(* Logix 5000 project; controller cal1615 1756-L62 rev 20.19; software revision 20.05; part 21 of 82 *)
(* tags used below, declared in another part *)
   AFI : BOOL;   // Always False Bit
   FAULT : BOOL;   // Fault AFI
   p01_param_fan_zero_speed : REAL;
   p01_param_open_oven_exh_sp : REAL;
   p01_recipe_active : recipe;   // Active Recipe
   p01r02 : routine;   // System Misc Control
   p01r09_open_oven : BOOL;
   p01r09_pb_global_reset : BOOL;   // System Modes PB: Global Fault Reset
   p02_dint_from_hmi : hmi_dint;
   p11_ai_exh_rpm : REAL;   // Zone 1 Analog Input Exhaust Fan RPM
   p11_ai_lfl : REAL;   // Zone 1 Analog Input Lower Flash Limit
   p11_ao_cv : REAL;   // Zone 1 Analog Output Control Valve
   p11_ao_exhaust_selected_speed : REAL;   // Zone 1 Analog Output Exhaust Fan VFD Selected Speed
   p11_di_burner_auto : BOOL;   // Zone 1 Digital Input Burner Auto
   p11_di_burner_safeties_ok : BOOL;   // Zone 1 Digital Input Burner Safeties Ok
   p11_di_door_open : BOOL;   // Zone 1 Digital Input Access Door Open
   p11_di_exh : acs800_di_normal;   // Zone 1 Digital Inputs Exhaust Fan
   p11_di_exh_fan_mtr_ts : BOOL;   // Zone 1 Digital Input Exhaust Fan Motor Thermostat OK
   p11_di_exh_flow_ok : BOOL;   // Zone 1 Digital Input Exhaust Flow OK
   p11_di_flame_failure : BOOL;   // Zone 1 Digital Input Flame Failure
   p11_di_flame_on : BOOL;   // Zone 1 Digital Input Burner is On
   p11_di_fresh_air_clean : BOOL;   // Zone 1 Digital Input Fresh Air Filter Dirty
   p11_di_high_limit_temp_ok : BOOL;   // Zone 1 Digital Input High Limit Temperature OK
   p11_di_recirc : acs800_di_normal;   // Zone 1 Digital Inputs Recirc Fan
   p11_di_recirc_flow_ok : BOOL;   // Zone 1 Digital Input Recirc Flow OK
   p11_di_sp00 : BOOL;   // Zone 1 Digital Input Recirculation Air Filter Dirty
   p11_di_sp1 : BOOL;
   p11_di_tc01_bo : BOOL;   // Zone 1 Digital Input Control Thermocouple 1 Failure
   p11_di_tc02_bo : BOOL;   // Zone 1 Digital Input Control Thermocouple 2 Failure
   p11_di_zone_air_clean : BOOL;   // Zone 1 Digital Input Combustion Air Filter Dirty
   p11_do_enable_burner : BOOL;   // Zone 1 Digital Output Enable Burner
   p11_do_exh : acs800_do_normal;   // Zone 1 Digital Output Exhaust Fan
   p11_do_rst_flame : BOOL;   // Zone 1 Digital Output Reset Flame Safety
   p11_param_lfl_hhl : REAL;   // Zone 1 Parameter High High Lower Flash Limit
   p11_param_lfl_hl : REAL;   // Zone 1 Parameter High LFL Limit
   p11_param_pid2_ff : REAL;   // Zone 1 Parameter Auto PID Bias
   p11_param_pid2_kd : REAL;   // Zone 1 Parameter Auto PID Derivative Gain
   p11_param_pid2_ki : REAL;   // Zone 1 Parameter Auto PID Integral Gain
   p11_param_pid2_kp : REAL;   // Zone 1 Parameter Auto PID Proportional Gain
   p11_param_tc01_dev : REAL;   // Zone 1 Parameter Oven Temperature Deviation from Setpoint
   p11_param_tc01_hl : REAL;   // Zone 1 Parameter Process Air High Limit
   p11r01 : routine;   // Zone 1 Main
   p11r02_shutdown_temp : BOOL;   // Zone 1 Misc Control Safe Shutdown Temperature
   p11r16_pid_temp_cv : DINT;   // Zone 1 Temperature Control Control Valve
   p11r16_temp_ok : BOOL;   // Zone 1 Temperature Control Temperature OK
   p11r20_safeties_ok : BOOL;   // Zone 1 Temperature Control Burner Safeties OK this Lightoff
   p11r20_state : DINT;   // Zone 1 Temperature Control State
   p11r30 : routine;   // Zone 1 Temperature Control
   p11r30_pb_zone_on : BOOL;   // Zone 1 Temperature Control PB: Start Zone Heat Control
   p11r30_pid_temp : PID;   // Zone 1 Temperature Control PID
   p11r30_pid_temp_pv : REAL;   // Zone 1 Temperature Control PID Temp Process Variable
   p11r30_pid_temp_sp_error : REAL;   // Zone 1 Temperature Control Setpoint/Process Variable Error (ABS)
   p11r30_request_deviation_warning : BOOL;   // Zone 1 Temperature Control Request Setpoint Deviation Warning
   p11r30_request_heat : BOOL;   // Zone 1 Temperature Control Request Heat
   p11r30_request_heat_last : BOOL;   // Zone 1 Temperature Control Request Heat Last Scan
   p11r30_request_manual : BOOL;   // Zone 1 Temperature Control Request Manual Control
   p11r30_request_soak_control : BOOL;   // Zone 1 Temperature Control Request Soak Control
   p11r30_timer_fault : TIMER[16];   // Zone 1 Temperature Control Fault Delay
   p11r30_timer_warning : TIMER[12];   // Zone 1 Temperature Control Warning Delay
   p11r31 : routine;   // Zone 1 Exhaust VFD
   p11r31_pb_start : BOOL;   // Zone 1 Exhaust VFD PB: Start
   p11r31_pb_stop : BOOL;   // Zone 1 Exhaust VFD PB: Stop
   p11r31_request_auto_run : BOOL;   // Zone 1 Exhaust Fan Run Request
   p11r31_run_permissive : BOOL;   // Zone 1 Exhaust VFD Run Permissive
   p11r31_timer_fault : TIMER[5];   // Zone 1 Exhaust VFD Fault Timer
   p11r31_timer_warning : TIMER[5];   // Zone 1 Exhaust VFD Waringing Timer
   p11r31_vfd_stopped : BOOL;   // Zone 1 Exhaust VFD VFD Stopped
   p11r32 : routine;   // Zone 1 Recirc VFD
   p12r30 : routine;   // Zone 2 Temperature Control
   p23_di_exhaust_speed_ok : BOOL;
   p23_di_supply_speed_ok : BOOL;
   p23r02 : routine;   // Impreg Misc Control
(* P11_Zone_1, continued *)

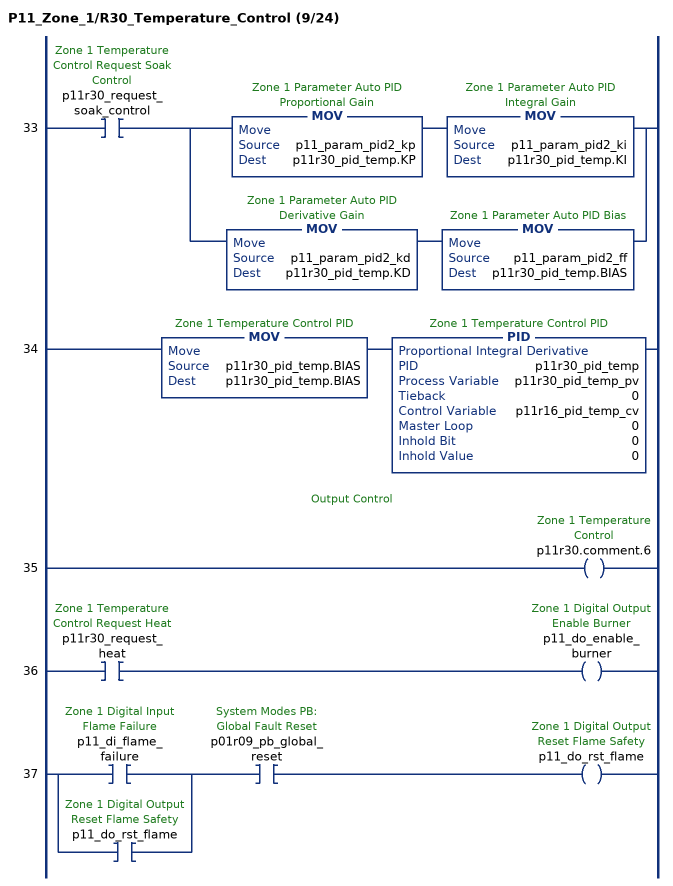
   [picture p329: P11_Zone_1/R30_Temperature_Control rungs 33-37]
   33: XIC(p11r30_request_soak_control)[MOV(p11_param_pid2_kp,p11r30_pid_temp.KP) MOV(p11_param_pid2_ki,p11r30_pid_temp.KI) ,MOV(p11_param_pid2_kd,p11r30_pid_temp.KD) MOV(p11_param_pid2_ff,p11r30_pid_temp.BIAS) ];
   34: MOV(p11r30_pid_temp.BIAS,p11r30_pid_temp.BIAS)PID(p11r30_pid_temp,p11r30_pid_temp_pv,0,p11r16_pid_temp_cv,0,0,0);
   // Output Control
   35: OTE(p11r30.comment.6);
   36: XIC(p11r30_request_heat)OTE(p11_do_enable_burner);
   37: [XIC(p11_di_flame_failure) ,XIC(p11_do_rst_flame) ]XIC(p01r09_pb_global_reset)OTE(p11_do_rst_flame);
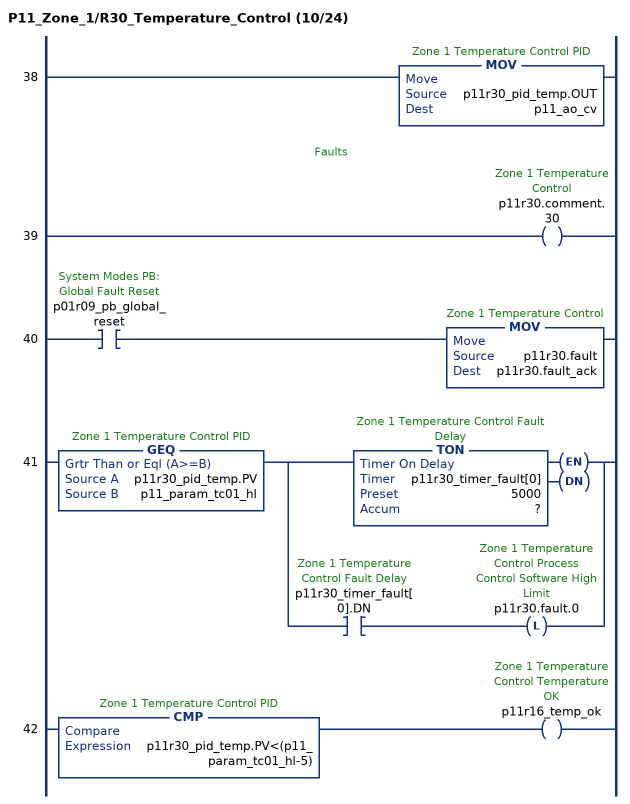
   38: MOV(p11r30_pid_temp.OUT,p11_ao_cv);
   // Faults
   39: OTE(p11r30.comment.30);
   40: XIC(p01r09_pb_global_reset)MOV(p11r30.fault,p11r30.fault_ack);
   41: GEQ(p11r30_pid_temp.PV,p11_param_tc01_hl)[TON(p11r30_timer_fault[0],?,?) ,XIC(p11r30_timer_fault[0].DN) OTL(p11r30.fault.0) ];
   42: CMP(p11r30_pid_temp.PV<(p11_param_tc01_hl-5))OTE(p11r16_temp_ok);
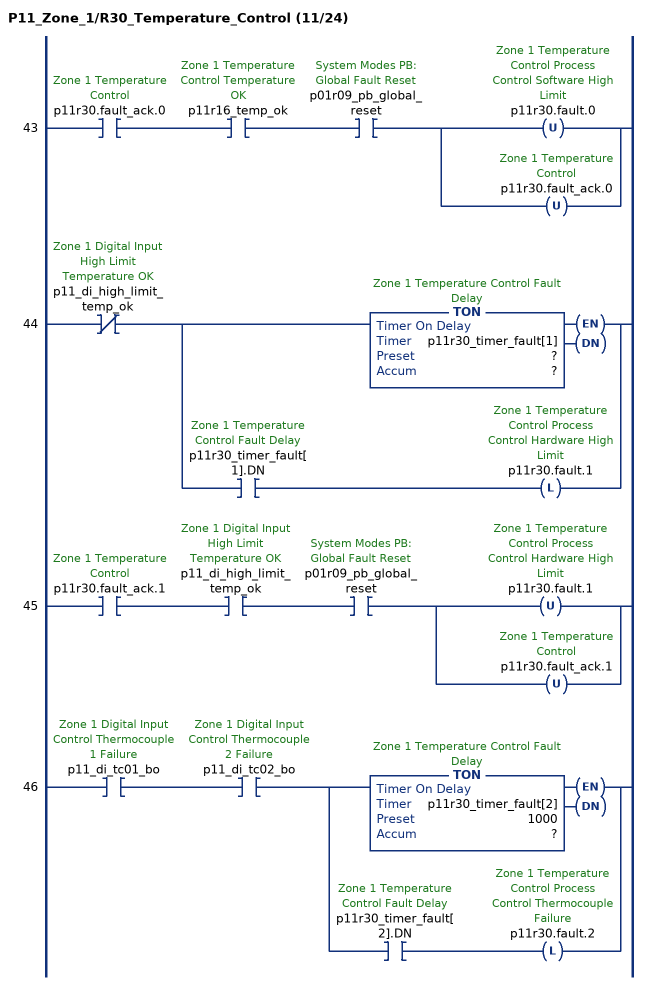
   43: XIC(p11r30.fault_ack.0)XIC(p11r16_temp_ok)XIC(p01r09_pb_global_reset)[OTU(p11r30.fault.0) ,OTU(p11r30.fault_ack.0) ];
   44: XIO(p11_di_high_limit_temp_ok)[TON(p11r30_timer_fault[1],?,?) ,XIC(p11r30_timer_fault[1].DN) OTL(p11r30.fault.1) ];
   45: XIC(p11r30.fault_ack.1)XIC(p11_di_high_limit_temp_ok)XIC(p01r09_pb_global_reset)[OTU(p11r30.fault.1) ,OTU(p11r30.fault_ack.1) ];
   46: XIC(p11_di_tc01_bo)XIC(p11_di_tc02_bo)[TON(p11r30_timer_fault[2],?,?) ,XIC(p11r30_timer_fault[2].DN) OTL(p11r30.fault.2) ];
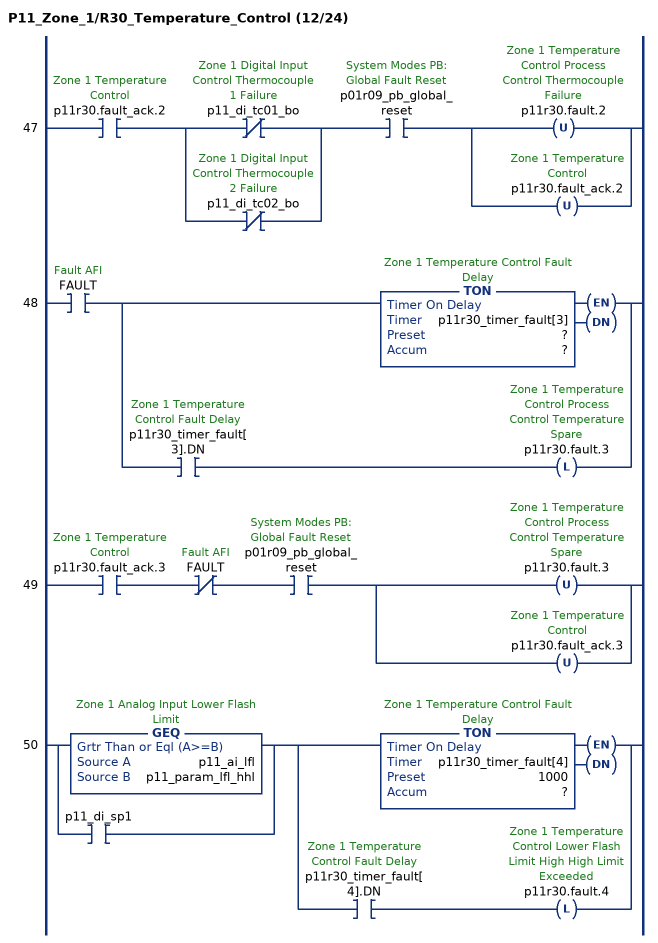
   47: XIC(p11r30.fault_ack.2)[XIO(p11_di_tc01_bo) ,XIO(p11_di_tc02_bo) ]XIC(p01r09_pb_global_reset)[OTU(p11r30.fault.2) ,OTU(p11r30.fault_ack.2) ];
   48: XIC(FAULT)[TON(p11r30_timer_fault[3],?,?) ,XIC(p11r30_timer_fault[3].DN) OTL(p11r30.fault.3) ];
   49: XIC(p11r30.fault_ack.3)XIO(FAULT)XIC(p01r09_pb_global_reset)[OTU(p11r30.fault.3) ,OTU(p11r30.fault_ack.3) ];
   50: [GEQ(p11_ai_lfl,p11_param_lfl_hhl) ,XIC(p11_di_sp1) ][TON(p11r30_timer_fault[4],?,?) ,XIC(p11r30_timer_fault[4].DN) OTL(p11r30.fault.4) ];
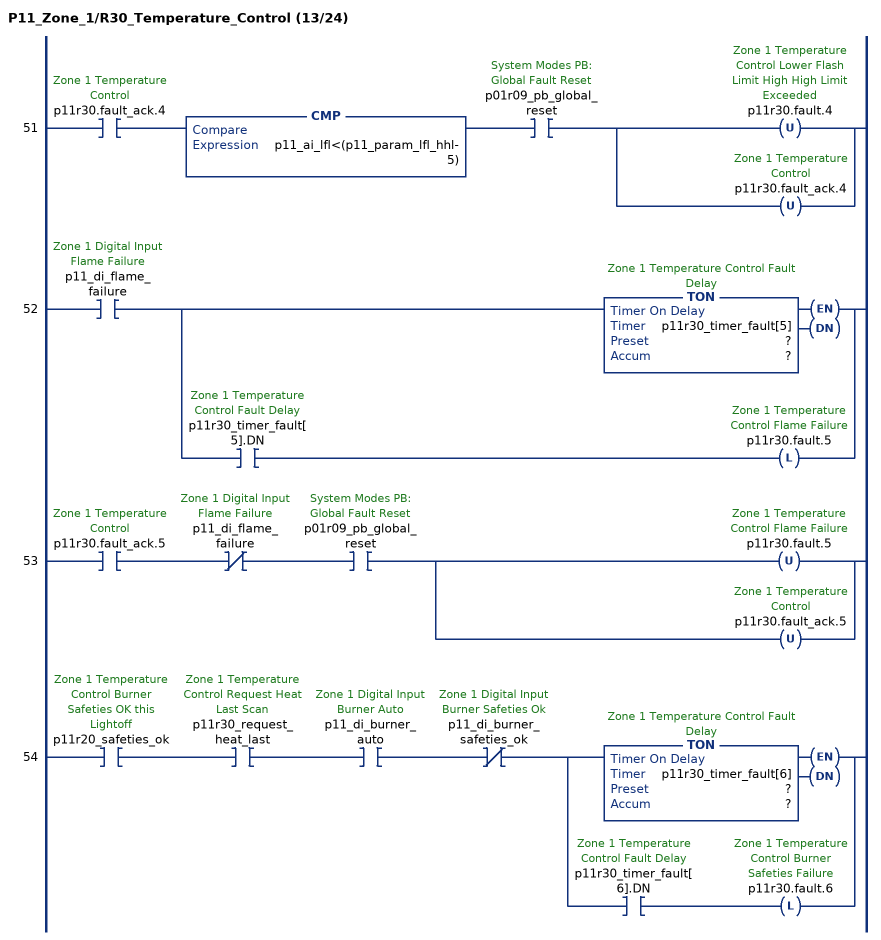
   51: XIC(p11r30.fault_ack.4)CMP(p11_ai_lfl<(p11_param_lfl_hhl-5))XIC(p01r09_pb_global_reset)[OTU(p11r30.fault.4) ,OTU(p11r30.fault_ack.4) ];
   52: XIC(p11_di_flame_failure)[TON(p11r30_timer_fault[5],?,?) ,XIC(p11r30_timer_fault[5].DN) OTL(p11r30.fault.5) ];
   53: XIC(p11r30.fault_ack.5)XIO(p11_di_flame_failure)XIC(p01r09_pb_global_reset)[OTU(p11r30.fault.5) ,OTU(p11r30.fault_ack.5) ];
   54: XIC(p11r20_safeties_ok)XIC(p11r30_request_heat_last)XIC(p11_di_burner_auto)XIO(p11_di_burner_safeties_ok)[TON(p11r30_timer_fault[6],?,?) ,XIC(p11r30_timer_fault[6].DN) OTL(p11r30.fault.6) ];
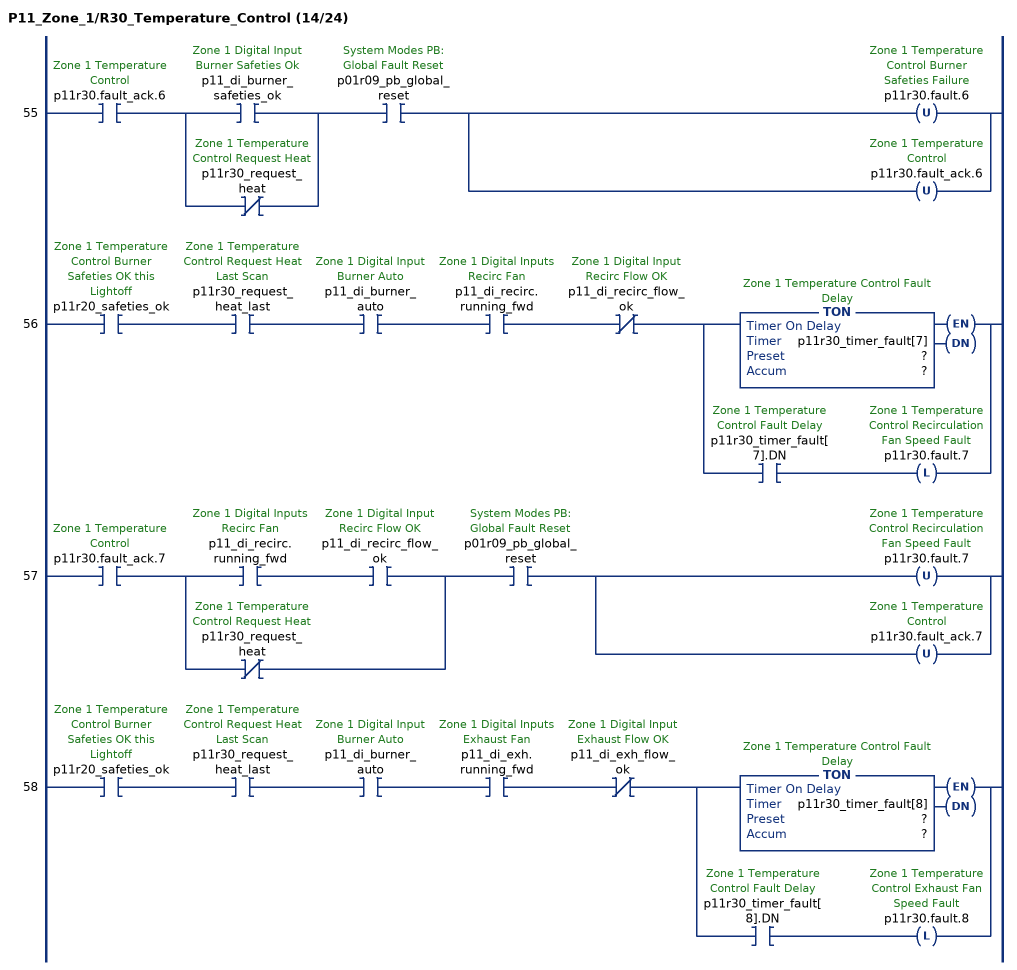
   55: XIC(p11r30.fault_ack.6)[XIC(p11_di_burner_safeties_ok) ,XIO(p11r30_request_heat) ]XIC(p01r09_pb_global_reset)[OTU(p11r30.fault.6) ,OTU(p11r30.fault_ack.6) ];
   56: XIC(p11r20_safeties_ok)XIC(p11r30_request_heat_last)XIC(p11_di_burner_auto)XIC(p11_di_recirc.running_fwd)XIO(p11_di_recirc_flow_ok)[TON(p11r30_timer_fault[7],?,?) ,XIC(p11r30_timer_fault[7].DN) OTL(p11r30.fault.7) ];
   57: XIC(p11r30.fault_ack.7)[XIC(p11_di_recirc.running_fwd) XIC(p11_di_recirc_flow_ok) ,XIO(p11r30_request_heat) ]XIC(p01r09_pb_global_reset)[OTU(p11r30.fault.7) ,OTU(p11r30.fault_ack.7) ];
   58: XIC(p11r20_safeties_ok)XIC(p11r30_request_heat_last)XIC(p11_di_burner_auto)XIC(p11_di_exh.running_fwd)XIO(p11_di_exh_flow_ok)[TON(p11r30_timer_fault[8],?,?) ,XIC(p11r30_timer_fault[8].DN) OTL(p11r30.fault.8) ];
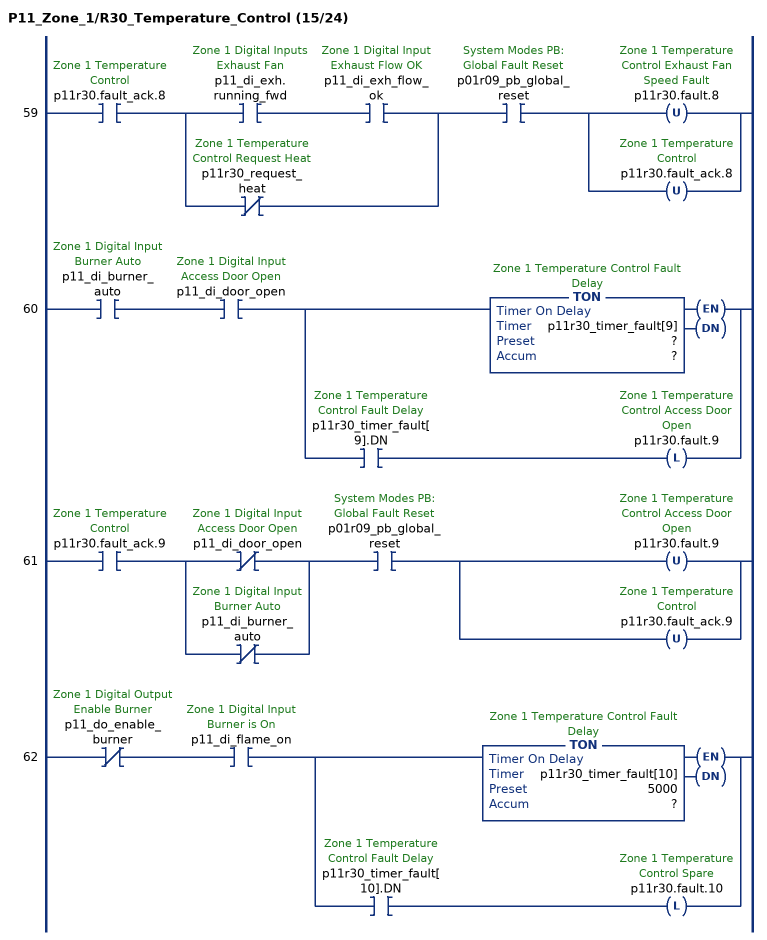
   59: XIC(p11r30.fault_ack.8)[XIC(p11_di_exh.running_fwd) XIC(p11_di_exh_flow_ok) ,XIO(p11r30_request_heat) ]XIC(p01r09_pb_global_reset)[OTU(p11r30.fault.8) ,OTU(p11r30.fault_ack.8) ];
   60: XIC(p11_di_burner_auto)XIC(p11_di_door_open)[TON(p11r30_timer_fault[9],?,?) ,XIC(p11r30_timer_fault[9].DN) OTL(p11r30.fault.9) ];
   61: XIC(p11r30.fault_ack.9)[XIO(p11_di_door_open) ,XIO(p11_di_burner_auto) ]XIC(p01r09_pb_global_reset)[OTU(p11r30.fault.9) ,OTU(p11r30.fault_ack.9) ];
   62: XIO(p11_do_enable_burner)XIC(p11_di_flame_on)[TON(p11r30_timer_fault[10],?,?) ,XIC(p11r30_timer_fault[10].DN) OTL(p11r30.fault.10) ];
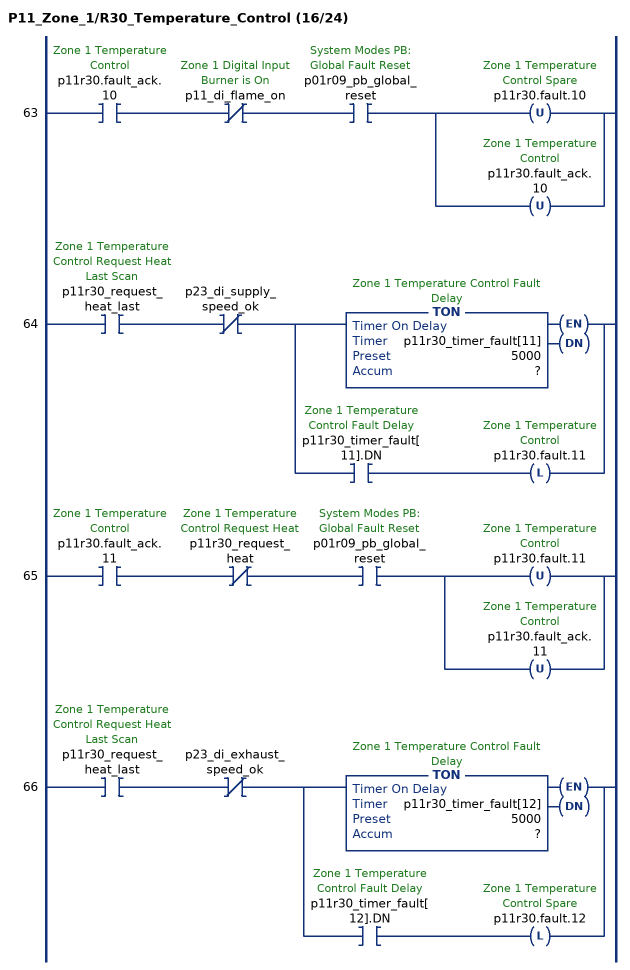
   63: XIC(p11r30.fault_ack.10)XIO(p11_di_flame_on)XIC(p01r09_pb_global_reset)[OTU(p11r30.fault.10) ,OTU(p11r30.fault_ack.10) ];
   64: XIC(p11r30_request_heat_last)XIO(p23_di_supply_speed_ok)[TON(p11r30_timer_fault[11],?,?) ,XIC(p11r30_timer_fault[11].DN) OTL(p11r30.fault.11) ];
   65: XIC(p11r30.fault_ack.11)XIO(p11r30_request_heat)XIC(p01r09_pb_global_reset)[OTU(p11r30.fault.11) ,OTU(p11r30.fault_ack.11) ];
   66: XIC(p11r30_request_heat_last)XIO(p23_di_exhaust_speed_ok)[TON(p11r30_timer_fault[12],?,?) ,XIC(p11r30_timer_fault[12].DN) OTL(p11r30.fault.12) ];
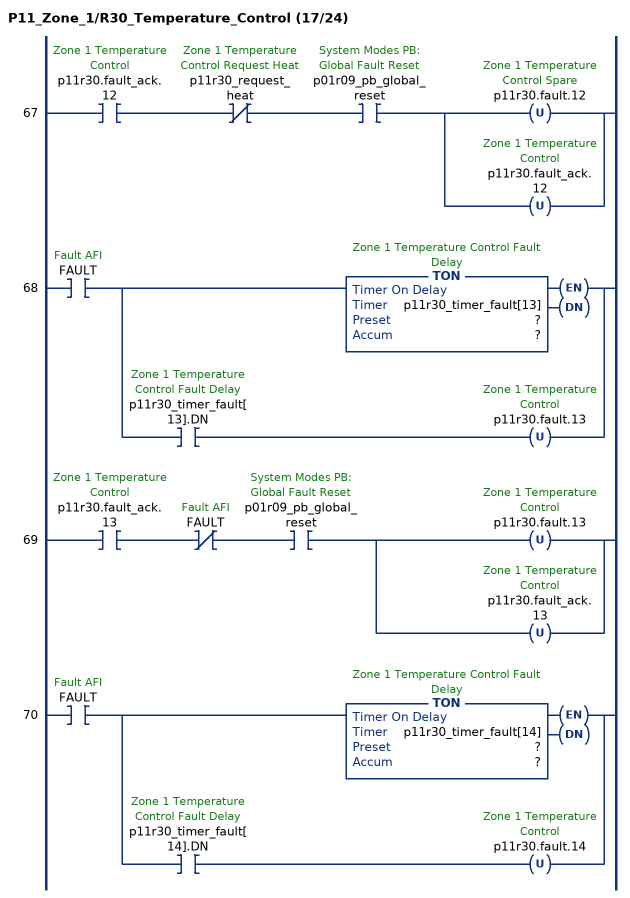
   67: XIC(p11r30.fault_ack.12)XIO(p11r30_request_heat)XIC(p01r09_pb_global_reset)[OTU(p11r30.fault.12) ,OTU(p11r30.fault_ack.12) ];
   68: XIC(FAULT)[TON(p11r30_timer_fault[13],?,?) ,XIC(p11r30_timer_fault[13].DN) OTU(p11r30.fault.13) ];
   69: XIC(p11r30.fault_ack.13)XIO(FAULT)XIC(p01r09_pb_global_reset)[OTU(p11r30.fault.13) ,OTU(p11r30.fault_ack.13) ];
   70: XIC(FAULT)[TON(p11r30_timer_fault[14],?,?) ,XIC(p11r30_timer_fault[14].DN) OTU(p11r30.fault.14) ];
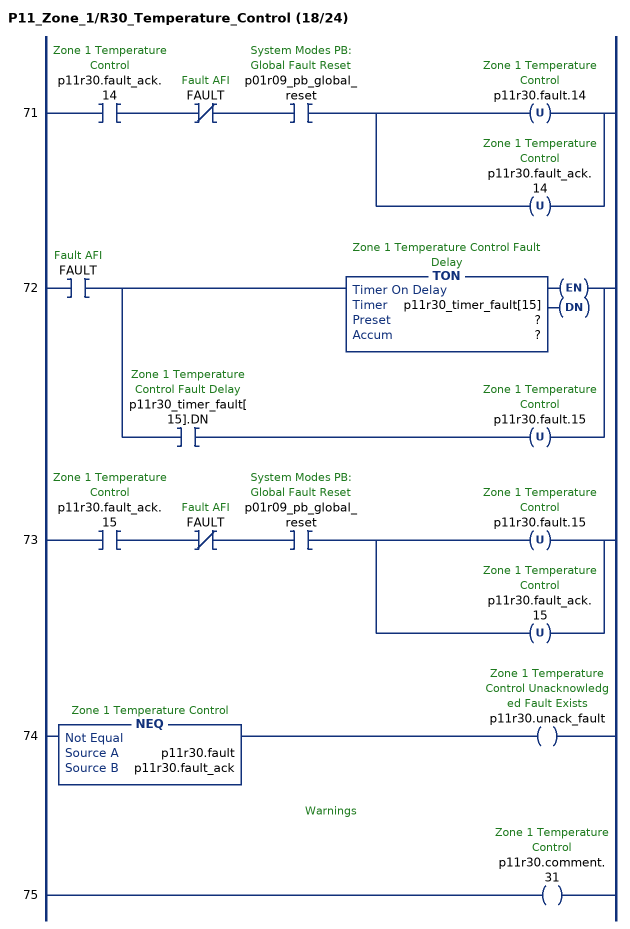
   71: XIC(p11r30.fault_ack.14)XIO(FAULT)XIC(p01r09_pb_global_reset)[OTU(p11r30.fault.14) ,OTU(p11r30.fault_ack.14) ];
   72: XIC(FAULT)[TON(p11r30_timer_fault[15],?,?) ,XIC(p11r30_timer_fault[15].DN) OTU(p11r30.fault.15) ];
   73: XIC(p11r30.fault_ack.15)XIO(FAULT)XIC(p01r09_pb_global_reset)[OTU(p11r30.fault.15) ,OTU(p11r30.fault_ack.15) ];
   74: NEQ(p11r30.fault,p11r30.fault_ack)OTE(p11r30.unack_fault);
   // Warnings
   75: OTE(p11r30.comment.31);
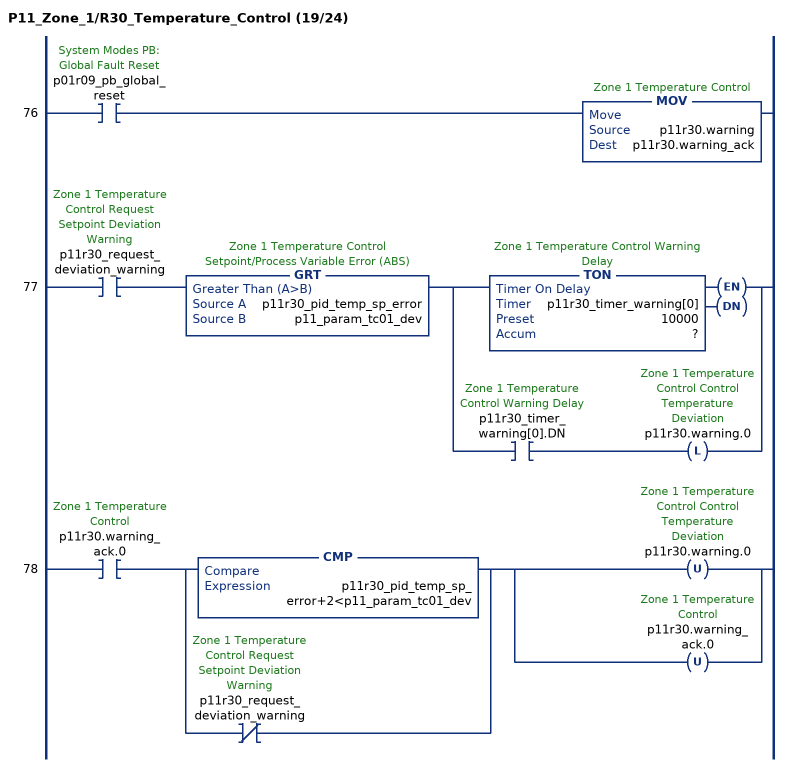
   76: XIC(p01r09_pb_global_reset)MOV(p11r30.warning,p11r30.warning_ack);
   77: XIC(p11r30_request_deviation_warning)GRT(p11r30_pid_temp_sp_error,p11_param_tc01_dev)[TON(p11r30_timer_warning[0],?,?) ,XIC(p11r30_timer_warning[0].DN) OTL(p11r30.warning.0) ];
   78: XIC(p11r30.warning_ack.0)[CMP(p11r30_pid_temp_sp_error+2<p11_param_tc01_dev) ,XIO(p11r30_request_deviation_warning) ][OTU(p11r30.warning.0) ,OTU(p11r30.warning_ack.0) ];
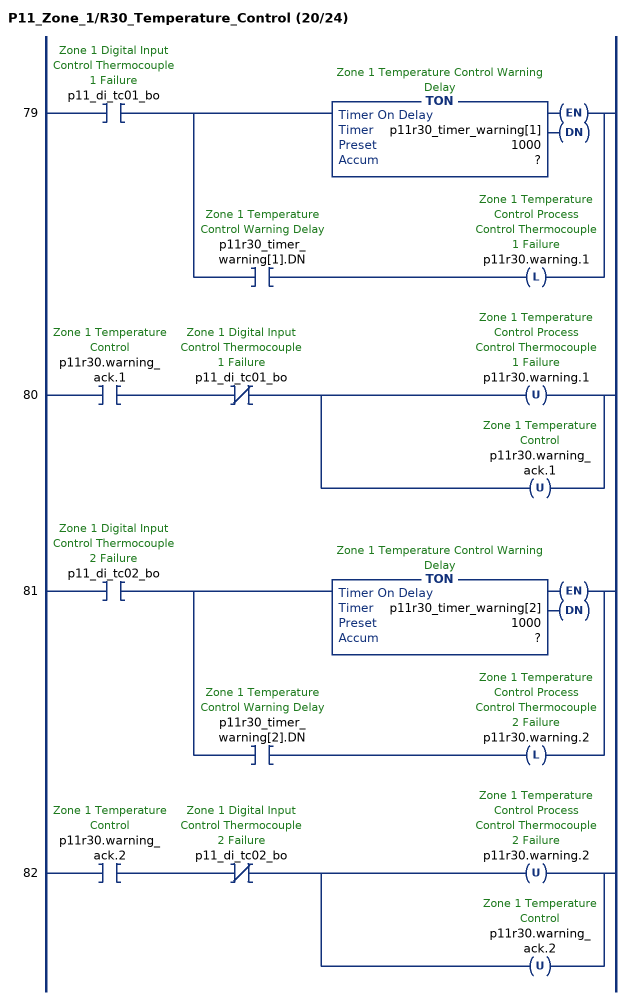
   79: XIC(p11_di_tc01_bo)[TON(p11r30_timer_warning[1],?,?) ,XIC(p11r30_timer_warning[1].DN) OTL(p11r30.warning.1) ];
   80: XIC(p11r30.warning_ack.1)XIO(p11_di_tc01_bo)[OTU(p11r30.warning.1) ,OTU(p11r30.warning_ack.1) ];
   81: XIC(p11_di_tc02_bo)[TON(p11r30_timer_warning[2],?,?) ,XIC(p11r30_timer_warning[2].DN) OTL(p11r30.warning.2) ];
   82: XIC(p11r30.warning_ack.2)XIO(p11_di_tc02_bo)[OTU(p11r30.warning.2) ,OTU(p11r30.warning_ack.2) ];
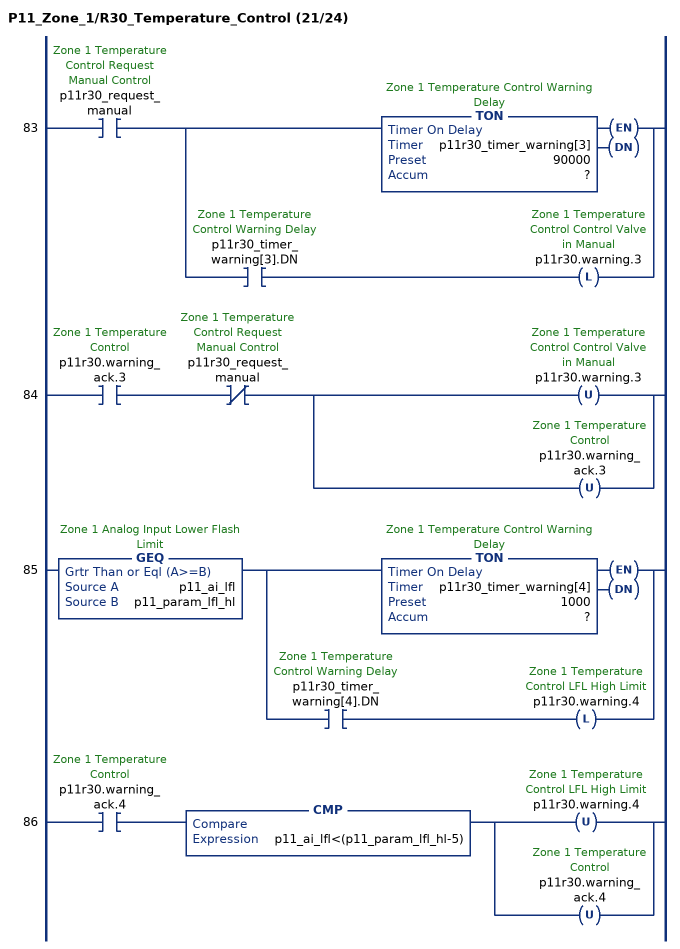
   83: XIC(p11r30_request_manual)[TON(p11r30_timer_warning[3],?,?) ,XIC(p11r30_timer_warning[3].DN) OTL(p11r30.warning.3) ];
   84: XIC(p11r30.warning_ack.3)XIO(p11r30_request_manual)[OTU(p11r30.warning.3) ,OTU(p11r30.warning_ack.3) ];
   85: GEQ(p11_ai_lfl,p11_param_lfl_hl)[TON(p11r30_timer_warning[4],?,?) ,XIC(p11r30_timer_warning[4].DN) OTL(p11r30.warning.4) ];
   86: XIC(p11r30.warning_ack.4)CMP(p11_ai_lfl<(p11_param_lfl_hl-5))[OTU(p11r30.warning.4) ,OTU(p11r30.warning_ack.4) ];
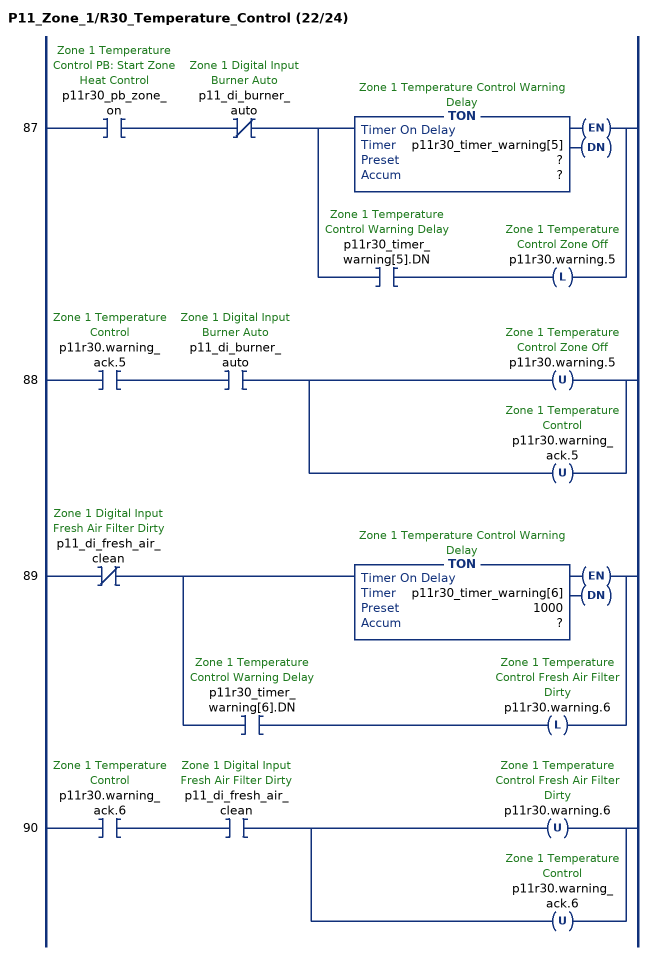
   87: XIC(p11r30_pb_zone_on)XIO(p11_di_burner_auto)[TON(p11r30_timer_warning[5],?,?) ,XIC(p11r30_timer_warning[5].DN) OTL(p11r30.warning.5) ];
   88: XIC(p11r30.warning_ack.5)XIC(p11_di_burner_auto)[OTU(p11r30.warning.5) ,OTU(p11r30.warning_ack.5) ];
   89: XIO(p11_di_fresh_air_clean)[TON(p11r30_timer_warning[6],?,?) ,XIC(p11r30_timer_warning[6].DN) OTL(p11r30.warning.6) ];
   90: XIC(p11r30.warning_ack.6)XIC(p11_di_fresh_air_clean)[OTU(p11r30.warning.6) ,OTU(p11r30.warning_ack.6) ];
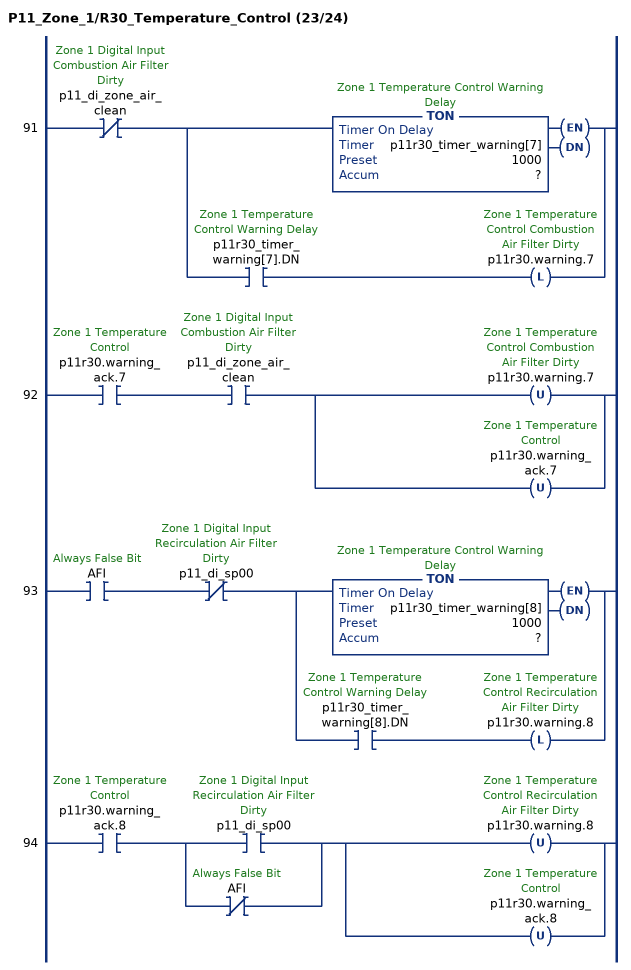
   91: XIO(p11_di_zone_air_clean)[TON(p11r30_timer_warning[7],?,?) ,XIC(p11r30_timer_warning[7].DN) OTL(p11r30.warning.7) ];
   92: XIC(p11r30.warning_ack.7)XIC(p11_di_zone_air_clean)[OTU(p11r30.warning.7) ,OTU(p11r30.warning_ack.7) ];
   93: XIC(AFI)XIO(p11_di_sp00)[TON(p11r30_timer_warning[8],?,?) ,XIC(p11r30_timer_warning[8].DN) OTL(p11r30.warning.8) ];
   94: XIC(p11r30.warning_ack.8)[XIC(p11_di_sp00) ,XIO(AFI) ][OTU(p11r30.warning.8) ,OTU(p11r30.warning_ack.8) ];
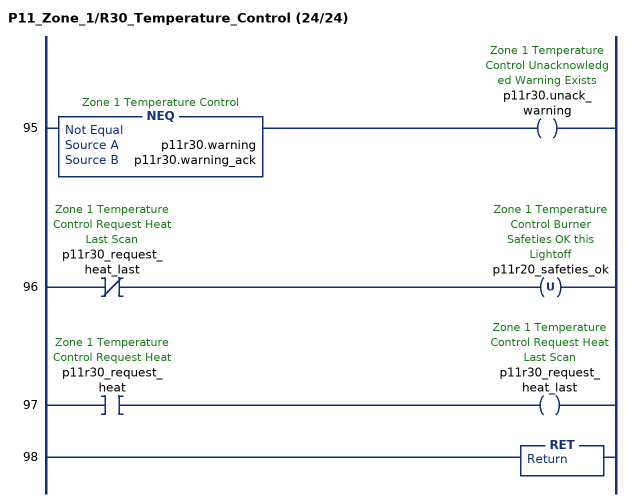
   95: NEQ(p11r30.warning,p11r30.warning_ack)OTE(p11r30.unack_warning);
   96: XIO(p11r30_request_heat_last)OTU(p11r20_safeties_ok);
   97: XIC(p11r30_request_heat)OTE(p11r30_request_heat_last);
   98: RET();
END_ROUTINE

ROUTINE R31_Exhaust_VFD   (* ladder *)
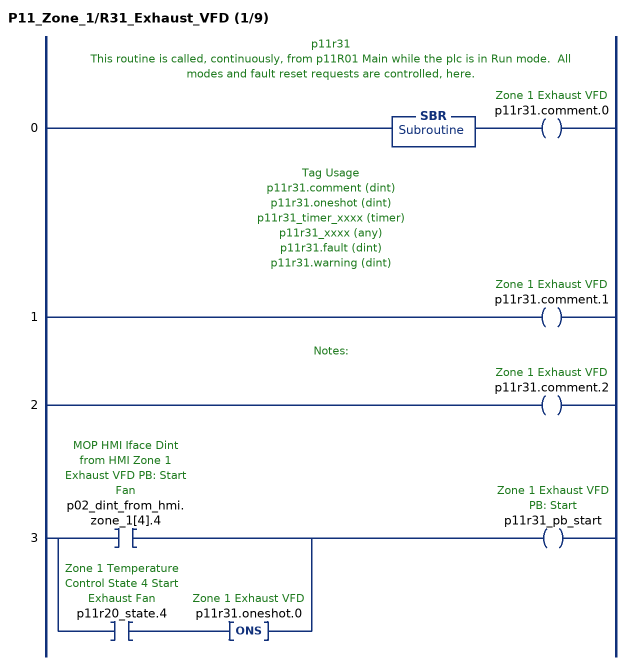
   // p11r31
   // This routine is called, continuously, from p11R01 Main while the plc is in Run mode.  All modes and fault reset requests are controlled, here.
   0: SBR()OTE(p11r31.comment.0);
   // Tag Usage
   // p11r31.comment (dint)
   // p11r31.oneshot (dint)
   // p11r31_timer_xxxx (timer)
   // p11r31_xxxx (any)
   // p11r31.fault (dint)
   // p11r31.warning (dint)
   1: OTE(p11r31.comment.1);
   // Notes:
   2: OTE(p11r31.comment.2);
   3: [XIC(p02_dint_from_hmi.zone_1[4].4) ,XIC(p11r20_state.4) ONS(p11r31.oneshot.0) ]OTE(p11r31_pb_start);
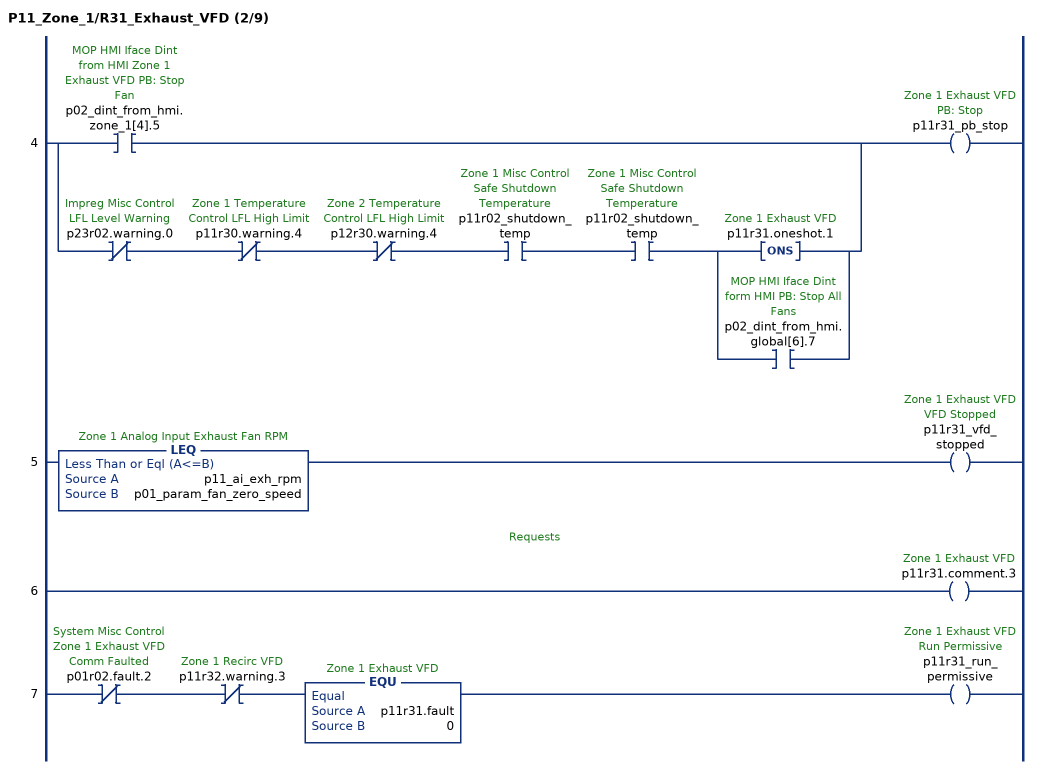
   4: [XIC(p02_dint_from_hmi.zone_1[4].5) ,XIO(p23r02.warning.0) XIO(p11r30.warning.4) XIO(p12r30.warning.4) XIC(p11r02_shutdown_temp) XIC(p11r02_shutdown_temp) [ONS(p11r31.oneshot.1) ,XIC(p02_dint_from_hmi.global[6].7) ] ]OTE(p11r31_pb_stop);
   5: LEQ(p11_ai_exh_rpm,p01_param_fan_zero_speed)OTE(p11r31_vfd_stopped);
   // Requests
   6: OTE(p11r31.comment.3);
   7: XIO(p01r02.fault.2)XIO(p11r32.warning.3)EQU(p11r31.fault,0)OTE(p11r31_run_permissive);
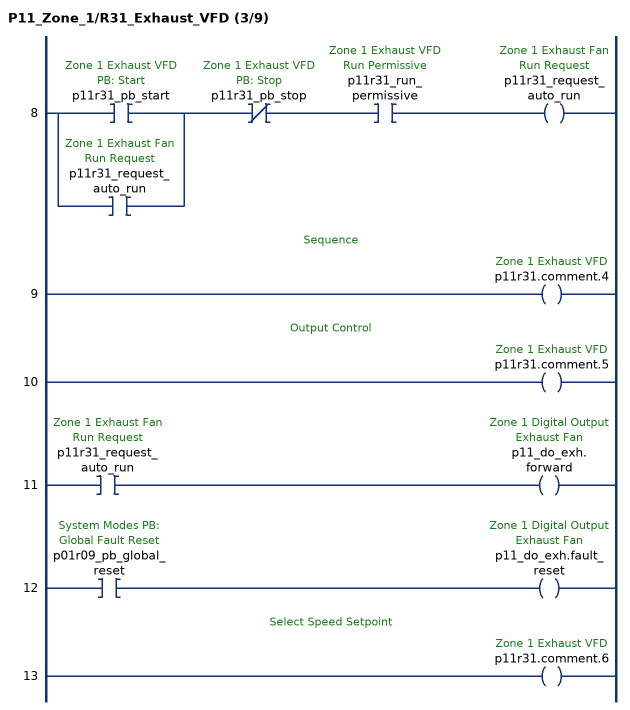
   8: [XIC(p11r31_pb_start) ,XIC(p11r31_request_auto_run) ]XIO(p11r31_pb_stop)XIC(p11r31_run_permissive)OTE(p11r31_request_auto_run);
   // Sequence
   9: OTE(p11r31.comment.4);
   // Output Control
   10: OTE(p11r31.comment.5);
   11: XIC(p11r31_request_auto_run)OTE(p11_do_exh.forward);
   12: XIC(p01r09_pb_global_reset)OTE(p11_do_exh.fault_reset);
   // Select Speed Setpoint
   13: OTE(p11r31.comment.6);
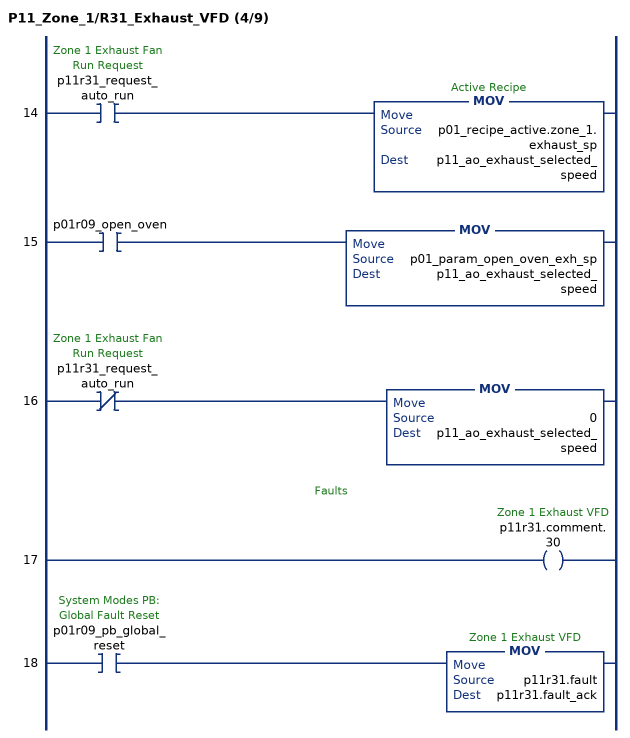
   14: XIC(p11r31_request_auto_run)MOV(p01_recipe_active.zone_1.exhaust_sp,p11_ao_exhaust_selected_speed);
   15: XIC(p01r09_open_oven)MOV(p01_param_open_oven_exh_sp,p11_ao_exhaust_selected_speed);
   16: XIO(p11r31_request_auto_run)MOV(0,p11_ao_exhaust_selected_speed);
   // Faults
   17: OTE(p11r31.comment.30);
   18: XIC(p01r09_pb_global_reset)MOV(p11r31.fault,p11r31.fault_ack);
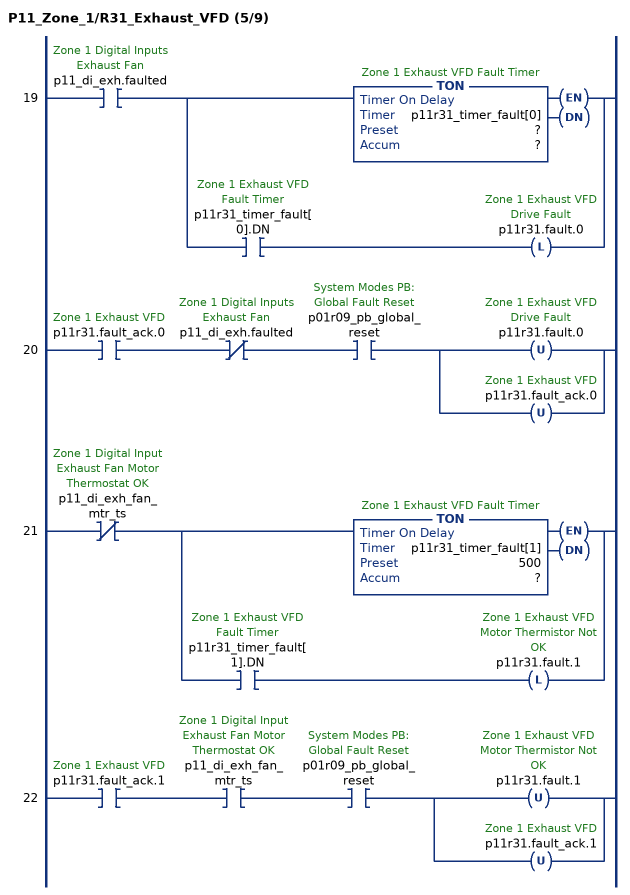
   19: XIC(p11_di_exh.faulted)[TON(p11r31_timer_fault[0],?,?) ,XIC(p11r31_timer_fault[0].DN) OTL(p11r31.fault.0) ];
   20: XIC(p11r31.fault_ack.0)XIO(p11_di_exh.faulted)XIC(p01r09_pb_global_reset)[OTU(p11r31.fault.0) ,OTU(p11r31.fault_ack.0) ];
   21: XIO(p11_di_exh_fan_mtr_ts)[TON(p11r31_timer_fault[1],?,?) ,XIC(p11r31_timer_fault[1].DN) OTL(p11r31.fault.1) ];
   22: XIC(p11r31.fault_ack.1)XIC(p11_di_exh_fan_mtr_ts)XIC(p01r09_pb_global_reset)[OTU(p11r31.fault.1) ,OTU(p11r31.fault_ack.1) ];
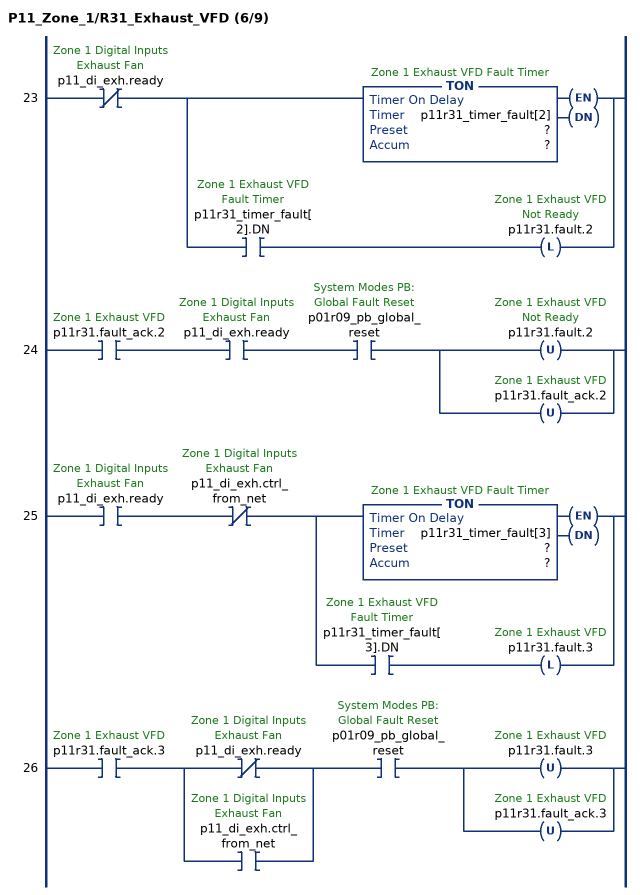
   23: XIO(p11_di_exh.ready)[TON(p11r31_timer_fault[2],?,?) ,XIC(p11r31_timer_fault[2].DN) OTL(p11r31.fault.2) ];
   24: XIC(p11r31.fault_ack.2)XIC(p11_di_exh.ready)XIC(p01r09_pb_global_reset)[OTU(p11r31.fault.2) ,OTU(p11r31.fault_ack.2) ];
   25: XIC(p11_di_exh.ready)XIO(p11_di_exh.ctrl_from_net)[TON(p11r31_timer_fault[3],?,?) ,XIC(p11r31_timer_fault[3].DN) OTL(p11r31.fault.3) ];
   26: XIC(p11r31.fault_ack.3)[XIO(p11_di_exh.ready) ,XIC(p11_di_exh.ctrl_from_net) ]XIC(p01r09_pb_global_reset)[OTU(p11r31.fault.3) ,OTU(p11r31.fault_ack.3) ];
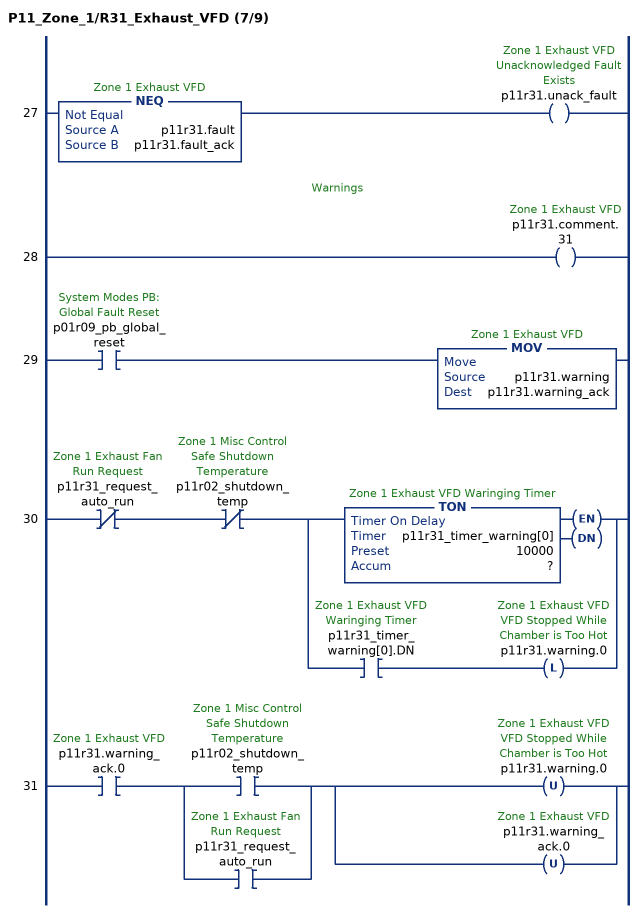
   27: NEQ(p11r31.fault,p11r31.fault_ack)OTE(p11r31.unack_fault);
   // Warnings
   28: OTE(p11r31.comment.31);
   29: XIC(p01r09_pb_global_reset)MOV(p11r31.warning,p11r31.warning_ack);
   30: XIO(p11r31_request_auto_run)XIO(p11r02_shutdown_temp)[TON(p11r31_timer_warning[0],?,?) ,XIC(p11r31_timer_warning[0].DN) OTL(p11r31.warning.0) ];
   31: XIC(p11r31.warning_ack.0)[XIC(p11r02_shutdown_temp) ,XIC(p11r31_request_auto_run) ][OTU(p11r31.warning.0) ,OTU(p11r31.warning_ack.0) ];
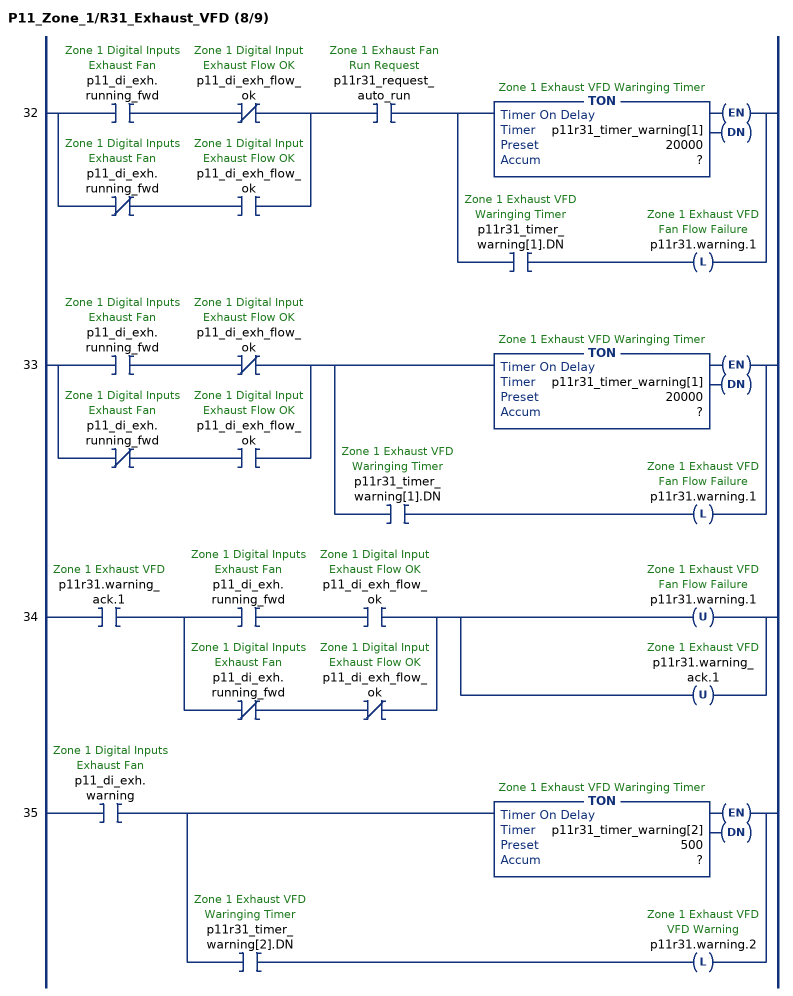
   32: [XIC(p11_di_exh.running_fwd) XIO(p11_di_exh_flow_ok) ,XIO(p11_di_exh.running_fwd) XIC(p11_di_exh_flow_ok) ]XIC(p11r31_request_auto_run)[TON(p11r31_timer_warning[1],?,?) ,XIC(p11r31_timer_warning[1].DN) OTL(p11r31.warning.1) ];
   33: [XIC(p11_di_exh.running_fwd) XIO(p11_di_exh_flow_ok) ,XIO(p11_di_exh.running_fwd) XIC(p11_di_exh_flow_ok) ][TON(p11r31_timer_warning[1],?,?) ,XIC(p11r31_timer_warning[1].DN) OTL(p11r31.warning.1) ];
   34: XIC(p11r31.warning_ack.1)[XIC(p11_di_exh.running_fwd) XIC(p11_di_exh_flow_ok) ,XIO(p11_di_exh.running_fwd) XIO(p11_di_exh_flow_ok) ][OTU(p11r31.warning.1) ,OTU(p11r31.warning_ack.1) ];
   35: XIC(p11_di_exh.warning)[TON(p11r31_timer_warning[2],?,?) ,XIC(p11r31_timer_warning[2].DN) OTL(p11r31.warning.2) ];
